// TIA Portal V20 export
TYPE "typeUnitCommunicationControlNode"
// stored: Namespace Unit1.Em13
   STRUCT
      ConveyorA { ExternalWritable := 'False'} : "Unit1.Em13.typeUnitCommunicationControlNodeConveyorA";
   END_STRUCT;
END_TYPE
